// TIA Portal V17 export
// export: Created 2025-03-07T09:16:53.2944181Z, ExportSetting WithDefaults, DisplayName Totally Integrated Automation Portal, DisplayVersion V17 Update 8, DisplayName TIA Portal Openness, DisplayVersion V17 Update 8, DisplayName TIA Portal Version Control Interface, DisplayVersion V17, DisplayName SINAMICS Startdrive Advanced, DisplayVersion V17 SP2, DisplayName SINAMICS Startdrive G110M, G120, G120C, G120D, G120P, G115D, DisplayVersion V17 SP2, DisplayName SINAMICS Startdrive G130, G150, S120, S150, SINAMICS MV, S210, DisplayVersion V17 SP2, DisplayName STEP 7 Professional, DisplayVersion V17 Update 8, DisplayName SINUMERIK ONE STEP 7 Toolbox, DisplayVersion V17 Update 12, DisplayName SINUMERIK 840D sl STEP 7 Toolbox, DisplayVersion V17 Update 12, DisplayName STEP 7 Safety, DisplayVersion V17 Update 6, DisplayName WinCC Advanced, DisplayVersion V17 Update 8
DATA_BLOCK "DB4001_FIXTURES_CALIBRATION"   // DB4001
{ S7_Optimized_Access := 'FALSE'; DB_Accessible_From_OPC_UA := 'FALSE' }
VERSION : 0.1
// stored: AutoNumber false, DBAccessibleFromOPCUA false, DBAccessibleFromWebserver true, IsOnlyStoredInLoadMemory false, IsWriteProtectedInAS false
   VAR
      FIXTURE_1_STA_2_CALIB_MEM : Bool;   // FIXTURE 1 STATION 2 CALIBRATION MEMORY
      FIXTURE_1_STA_3_CALIB_MEM : Bool;   // FIXTURE 1 STATION 3 CALIBRATION MEMORY
      FIXTURE_2_STA_2_CALIB_MEM : Bool;   // FIXTURE 2 STATION 2 CALIBRATION MEMORY
      FIXTURE_2_STA_3_CALIB_MEM : Bool;   // FIXTURE 2 STATION 3 CALIBRATION MEMORY
      FIXTURE_3_STA_2_CALIB_MEM : Bool;   // FIXTURE 3 STATION 2 CALIBRATION MEMORY
      FIXTURE_3_STA_3_CALIB_MEM : Bool;   // FIXTURE 3 STATION 3 CALIBRATION MEMORY
      FIXTURE_4_STA_2_CALIB_MEM : Bool;   // FIXTURE 4 STATION 2 CALIBRATION MEMORY
      FIXTURE_4_STA_3_CALIB_MEM : Bool;   // FIXTURE 4 STATION 3 CALIBRATION MEMORY
      ALL_FIXTURES_STA_2_CALIB_MEM : Bool;   // ALL FIXTURES STATION 2 CALIBRATION MEMORY
      ALL_FIXTURES_STA_3_CALIB_MEM : Bool;   // ALL FIXTURES STATION 3 CALIBRATION MEMORY
      ALL_FIXTURES_CALIB_MEM : Bool;   // ALL FIXTURES CALIBRATION MEMORY DONE
   END_VAR
BEGIN
END_DATA_BLOCK
